/// Function convert EtherCat device state from a slave into an text
FUNCTION F_Diagnostic_EcDeviceState : WSTRING(80)
VAR_INPUT
	/// Function input
	nDeviceState			:BYTE;
END_VAR
VAR
END_VAR

CASE nDeviceState OF
	EC_DEVICE_STATE_INIT:
		F_Diagnostic_EcDeviceState := "EtherCat Device State: INIT";
		
	EC_DEVICE_STATE_PREOP:
		F_Diagnostic_EcDeviceState := "EtherCat Device State: Pre-Operational";
		
	EC_DEVICE_STATE_BOOTSTRAP:
		F_Diagnostic_EcDeviceState := "EtherCat Device State: Bootstrap";
		
	EC_DEVICE_STATE_SAFEOP:
		F_Diagnostic_EcDeviceState := "EtherCat Device State: Safe-Operational";
		
	EC_DEVICE_STATE_OP:
		F_Diagnostic_EcDeviceState := "EtherCat Device State: Operational";
		
	EC_DEVICE_STATE_ERROR:
		F_Diagnostic_EcDeviceState := "EtherCat Device State: Statemachine-error in slave";
		
	EC_DEVICE_STATE_INVALID_VPRS:
		F_Diagnostic_EcDeviceState := "EtherCat Device State: Invalid VendorID, Productcode, revisionnumber or serialnumber";
		
	EC_DEVICE_STATE_INITCMD_ERROR:
		F_Diagnostic_EcDeviceState := "EtherCat Device State: INIT command error";
		
	ELSE 
		F_Diagnostic_EcDeviceState := "EtherCat Device State: Undefined";
END_CASE

END_FUNCTION

(* stored: Version 1.1.0.1, ProductVersion 3.1.4024.11
   POU F_Diagnostic_EcDeviceState: Id {521f43c6-1593-4734-8f55-2cafc7884e56}, SpecialFunc None *)
